INTERFACE I_AliasDatatypeAddedEvent EXTENDS I_Event

PROPERTY PUBLIC Target : I_AliasDatatype
GET
END_GET
END_PROPERTY

END_INTERFACE

(* stored: Version 1.1.0.1, ProductVersion 3.1.4024.12
   Itf I_AliasDatatypeAddedEvent: Id {ab4ea38b-d4f3-0068-3436-6fc4a05e8994}
   Property Target: Id {fb95e671-7ff9-0bd3-16d6-abec709b918d}
   Get Get: Id {b2743876-f7f2-0468-18a7-1e881f176b5f} *)
